FUNCTION GENERATE_FILENAME : STRING
VAR_INPUT
	sPrefix : STRING;
	stTime : TIMESTRUCT;
	sSuffix : STRING;
END_VAR
VAR
	sOutput : STRING;
	sTime : STRING;
END_VAR

sTime := SYSTEMTIME_TO_STRING(stTime);

sOutput := sPrefix;

//sOutput := CONCAT(sOutput, 'test');

sOutput := CONCAT(sOutput, LEFT(sTime, 10));

sOutput := CONCAT(sOutput, ' ');
sOutput := CONCAT(sOutput, MID(sTime, 2, 12));
sOutput := CONCAT(sOutput, '-');
sOutput := CONCAT(sOutput, MID(sTime, 2, 15));
sOutput := CONCAT(sOutput, '-');
sOutput := CONCAT(sOutput, MID(sTime, 2, 18));

sOutput := CONCAT(sOutput, sSuffix);

GENERATE_FILENAME := sOutput;

END_FUNCTION

(* stored: Version 1.1.0.1, ProductVersion 3.1.4022.10
   POU GENERATE_FILENAME: Id {5a3f84cf-3117-47c3-8621-861ae5392137}, SpecialFunc None *)
